Universal Robots PolyScope program: learning_shifting_for_grasping.urp

Program learning_shifting_for_grasping (installation=default directory=/programs createdIn=5.9.1.1031110 lastSavedIn=5.9.1.1031110 robotSerialNumber=20185500256)
Calibrated DH parameters: a=[0.000163, -0.146131, -0.38577, 0.000126, -0.000021, 0]; d=[0.161954, 188.306531, -157.478086, -30.695088, 0.099716, 0.099628]; alpha=[1.569701, -0.00212, 0.002263, 1.570438, -1.570123, 0]; deltaTheta=[0, -1.219859, 7.681919, -0.178877, -0.000001, 0]
InitVariablesNode variables(variable(name=reached_point, expression=False))
BeforeStart
  Call URCancelManualMove
  SuppressedNode
    Call InitGripper
  MoveJ speed 60 deg/s, acceleration 80 deg/s^2 (useActiveTCP=true) feature=Base
    Waypoint HomeWP: TCP in base x=132.769 y=-491.632 z=236.295 mm, rx=0.0018 ry=-3.1384 rz=0.0008 rad; joints [90.004, -89.995, 90.002, -89.997, -90.004, 0.023] deg; TCP offset x=0 y=0 z=250.5 mm, rx=0 ry=0 rz=0 rad
Robot Program (runOnlyOnce=false)
  MoveJ speed 60 deg/s, acceleration 80 deg/s^2 (useActiveTCP=true) feature=Base
    Waypoint Waypoint (Variable): variable(featureName=cam_bin1)
  GripperWidth := 0
  Call SetGripperWidth
  Call MoveToApproach
  Call MoveToGrasp
  URCap EGI Grip (SCHUNK Gripper EGI for UR, SCHUNK GmbH & Co.) dataModel(position=32.5, position_tol=0.5, dummy=0.5, use_work_piece=true, async_exe=true, grip_type=0)
  If egiGripped()
    Call MoveToSafety
    MoveJ speed 60 deg/s, acceleration 80 deg/s^2 (useActiveTCP=true) feature=Base
      Waypoint Waypoint (Variable): variable(featureName=cam_bin2)
    URCap EGI Grip (SCHUNK Gripper EGI for UR, SCHUNK GmbH & Co.) dataModel(grip_type=3)
  Else 
    GripperWidth := 1
    Call SetGripperWidth
    MoveJ speed 60 deg/s, acceleration 80 deg/s^2 (useActiveTCP=true) feature=Base
      Waypoint Waypoint (Variable): variable(featureName=cam_bin1)
  SuppressedNode
    Call MoveToSafety
SubProgram  [hidden by the author, left out]
SubProgram  [hidden by the author, left out]
SubProgram  [hidden by the author, left out]
SubProgram  [hidden by the author, left out]
SubProgram  [hidden by the author, left out]
SubProgram  [hidden by the author, left out]
SubProgram URCancelManualMove [hidden by the author, left out]
SubProgram InitGripper [hidden by the author, left out]
SubProgram SetGripperWidth [hidden by the author, left out]
SubProgram MoveToApproach [hidden by the author, left out]
SubProgram MoveToGrasp [hidden by the author, left out]
SubProgram MoveToSafety [hidden by the author, left out]
